TEXTLIST S1_Warnings
  0 = 'Station 1 Warning'
  1 = 'Warning 2'
  2 = 'Warning 3'
  3 = 'Low Oil Level'
   = ''
END_TEXTLIST

(* stored: Version 1.1.0.1, ProductVersion 3.1.4024.12
   TextList S1_Warnings: Id {96d2cb34-4440-0f22-1983-5a68db06ade9} *)
